// TwinCAT 3 PLC project ScatterSlits
// ProgramVersion: 3.1.4022.3
// libraries:
//   Tc2_MC2, * (Beckhoff Automation GmbH)
//   Tc2_Standard, * (Beckhoff Automation GmbH)
//   Tc2_System, * (Beckhoff Automation GmbH)
//   Tc3_Module, * (Beckhoff Automation GmbH)
// project tree:
//   DUTs/ DUT_M.TcDUT, E_HomeState.TcDUT (not stored), MoveState_t.TcDUT
//   / PlcTask.TcTTO
//   POUs/ FB_Home.TcPOU, FB_HomeToSwitch.TcPOU, FB_Motion.TcPOU, MAIN.TcPOU
// real-time tasks:
//   TASK PlcTask: cycle T#10ms, priority 20, ADS port 350
// motion (NC):
//   TASK NC-Task 1 SAF: cycle T#2ms, priority 4, ADS port 501
//   TASK NC-Task 1 SVB: cycle T#10ms, priority 8, ADS port 511
//   AXIS Axis 1 (id 1)
//     Velo: Maximum=2.2
//     OtherSettings: AllowMotionCmdToSlave=true
//     encoder EncType=4
//       EncPara: MaxCount=#x0000ffff
//         SoftEndMinControl: Range=0.05
//         Inc: RefSoftSyncMask=#x0000ffff
//     drive DrvType=24
//       Analog: VeloReferenz=2, ScaleFactorActTorque=0.1
//       TimeComp: TaskDelayCycles=1
//     controller CtrType=1
//       CtrPara: PriorControlFactor=1
//         PosDiffControl: Range=0.05
//         Observer: BandWidth=20
//   AXIS Axis 2 (id 2)
//     Velo: Maximum=2.2
//     OtherSettings: AllowMotionCmdToSlave=true
//     encoder EncType=4
//       EncPara: Inverse=true, MaxCount=#x0000ffff
//         Inc: RefSoftSyncMask=#x0000ffff
//     drive DrvType=24
//       Analog: VeloReferenz=2, ScaleFactorActTorque=0.1
//       TimeComp: TaskDelayCycles=1
//     controller CtrType=1
//       CtrPara: PriorControlFactor=1
//         PosDiffControl: Range=0.05
//         Observer: BandWidth=20
//   AXIS Axis 3 (id 3)
//     Velo: Maximum=2.2
//     OtherSettings: AllowMotionCmdToSlave=true
//     encoder EncType=4
//       EncPara: Inverse=true, MaxCount=#x0000ffff
//         Inc: RefSoftSyncMask=#x0000ffff
//     drive DrvType=24
//       Analog: VeloReferenz=2, ScaleFactorActTorque=0.1
//       TimeComp: TaskDelayCycles=1
//     controller CtrType=1
//       CtrPara: PriorControlFactor=1
//         PosDiffControl: Range=0.1
//         Observer: BandWidth=20
//   AXIS Axis 4 (id 4)
//     Velo: Maximum=2.2
//     OtherSettings: AllowMotionCmdToSlave=true
//     encoder EncType=4
//       EncPara: MaxCount=#x0000ffff
//         Inc: RefSoftSyncMask=#x0000ffff
//     drive DrvType=24
//       Analog: VeloReferenz=2, ScaleFactorActTorque=0.1
//       TimeComp: TaskDelayCycles=1
//     controller CtrType=1
//       CtrPara: PriorControlFactor=1
//         PosDiffControl: Range=0.1
//         Observer: BandWidth=20
// I/O:
//   DEVICE Device 1 (EtherCAT), AmsNetId 134.79.81.23.2.1
//     Term 1 (EK1100) [EK1100 EtherCAT Coupler (2A E-Bus)]
//       M1  (EL7031) [EL7031 1Ch. Stepper motor output stage (24V, 1.5A)]
//       E1(EL5101) [EL5101 1Ch. Inc. Encoder 5V]
//       M2 (EL7031) [EL7031 1Ch. Stepper motor output stage (24V, 1.5A)]
//       E2 (EL5101) [EL5101 1Ch. Inc. Encoder 5V]
//       M3 (EL7031) [EL7031 1Ch. Stepper motor output stage (24V, 1.5A)]
//       E3 (EL5101) [EL5101 1Ch. Inc. Encoder 5V]
//       M4 (EL7031) [EL7031 1Ch. Stepper motor output stage (24V, 1.5A)]
//       E4 (EL5101) [EL5101 1Ch. Inc. Encoder 5V]
//       Term 10 (EL9011) [EL9011 End Terminal]
// variable links:
//   NC-Task 1 SAF/Axes/Axis 1 <-> Device 1 (EtherCAT)/Term 1 (EK1100)/E1(EL5101)
//     Enc/Inputs/In/nDataIn1[0] <-> ENC Status compact/Counter value
//     Enc/Inputs/In/nDataIn2[0] <-> ENC Status compact/Latch value
//     Enc/Inputs/In/nState1 @bit 4 <-> ENC Status compact/Status/Counter overflow
//     Enc/Inputs/In/nState1 @bit 3 <-> ENC Status compact/Status/Counter underflow
//     Enc/Inputs/In/nState1 @bit 7 <-> ENC Status compact/Status/Extrapolation stall
//     Enc/Inputs/In/nState1 <-> ENC Status compact/Status/Latch C valid
//     Enc/Inputs/In/nState1 @bit 1 <-> ENC Status compact/Status/Latch extern valid
//     Enc/Inputs/In/nState1 @bit 6 <-> ENC Status compact/Status/Open circuit
//     Enc/Inputs/In/nState1 @bit 2 <-> ENC Status compact/Status/Set counter done
//     Enc/Inputs/In/nState1 @bit 5 <-> ENC Status compact/Status/Status of input status
//     Enc/Inputs/In/nState2 @bit 4 <-> ENC Status compact/Status/Status of extern latch
//     Enc/Inputs/In/nState2 <-> ENC Status compact/Status/Status of input A
//     Enc/Inputs/In/nState2 @bit 1 <-> ENC Status compact/Status/Status of input B
//     Enc/Inputs/In/nState2 @bit 2 <-> ENC Status compact/Status/Status of input C
//     Enc/Inputs/In/nState2 @bit 3 <-> ENC Status compact/Status/Status of input gate
//     Enc/Inputs/In/nState2 @bit 5 <-> ENC Status compact/Status/Sync error
//     Enc/Inputs/In/nState2 @bit 6 <-> ENC Status compact/Status/TxPDO State
//     Enc/Inputs/In/nState2 @bit 7 <-> ENC Status compact/Status/TxPDO Toggle
//     Enc/Inputs/In/nState4 @bit 1 <-> WcState/InputToggle
//     Enc/Inputs/In/nState4 <-> WcState/WcState
//     Enc/Outputs/Out/nCtrl1 <-> ENC Control compact/Control/Enable latch C
//     Enc/Outputs/Out/nCtrl1 @bit 3 <-> ENC Control compact/Control/Enable latch extern on negative edge
//     Enc/Outputs/Out/nCtrl1 @bit 1 <-> ENC Control compact/Control/Enable latch extern on positive edge
//     Enc/Outputs/Out/nCtrl1 @bit 2 <-> ENC Control compact/Control/Set counter
//     Enc/Outputs/Out/nDataOut1[0] <-> ENC Control compact/Set counter value
//   NC-Task 1 SAF/Axes/Axis 1 <-> Device 1 (EtherCAT)/Term 1 (EK1100)/M1  (EL7031)
//     Drive/Inputs/In/nState1 @bit 3 <-> STM Status/Status/Error
//     Drive/Inputs/In/nState1 @bit 5 <-> STM Status/Status/Moving negative
//     Drive/Inputs/In/nState1 @bit 4 <-> STM Status/Status/Moving positive
//     Drive/Inputs/In/nState1 @bit 1 <-> STM Status/Status/Ready
//     Drive/Inputs/In/nState1 <-> STM Status/Status/Ready to enable
//     Drive/Inputs/In/nState1 @bit 6 <-> STM Status/Status/Torque reduced
//     Drive/Inputs/In/nState1 @bit 2 <-> STM Status/Status/Warning
//     Drive/Inputs/In/nState2 @bit 5 <-> STM Status/Status/Sync error
//     Drive/Inputs/In/nState2 @bit 7 <-> STM Status/Status/TxPDO Toggle
//     Drive/Inputs/In/nState4 @bit 1 <-> WcState/InputToggle
//     Drive/Inputs/In/nState4 <-> WcState/WcState
//     Drive/Outputs/Out/nCtrl1 <-> STM Control/Control/Enable
//     Drive/Outputs/Out/nCtrl1 @bit 2 <-> STM Control/Control/Reduce torque
//     Drive/Outputs/Out/nCtrl1 @bit 1 <-> STM Control/Control/Reset
//     Drive/Outputs/Out/nDataOut2[0] <-> STM Velocity/Velocity
//   NC-Task 1 SAF/Axes/Axis 2 <-> Device 1 (EtherCAT)/Term 1 (EK1100)/E2 (EL5101)
//     Enc/Inputs/In/nDataIn1[0] <-> ENC Status compact/Counter value
//     Enc/Inputs/In/nDataIn2[0] <-> ENC Status compact/Latch value
//     Enc/Inputs/In/nState1 @bit 4 <-> ENC Status compact/Status/Counter overflow
//     Enc/Inputs/In/nState1 @bit 3 <-> ENC Status compact/Status/Counter underflow
//     Enc/Inputs/In/nState1 @bit 7 <-> ENC Status compact/Status/Extrapolation stall
//     Enc/Inputs/In/nState1 <-> ENC Status compact/Status/Latch C valid
//     Enc/Inputs/In/nState1 @bit 1 <-> ENC Status compact/Status/Latch extern valid
//     Enc/Inputs/In/nState1 @bit 6 <-> ENC Status compact/Status/Open circuit
//     Enc/Inputs/In/nState1 @bit 2 <-> ENC Status compact/Status/Set counter done
//     Enc/Inputs/In/nState1 @bit 5 <-> ENC Status compact/Status/Status of input status
//     Enc/Inputs/In/nState2 @bit 4 <-> ENC Status compact/Status/Status of extern latch
//     Enc/Inputs/In/nState2 <-> ENC Status compact/Status/Status of input A
//     Enc/Inputs/In/nState2 @bit 1 <-> ENC Status compact/Status/Status of input B
//     Enc/Inputs/In/nState2 @bit 2 <-> ENC Status compact/Status/Status of input C
//     Enc/Inputs/In/nState2 @bit 3 <-> ENC Status compact/Status/Status of input gate
//     Enc/Inputs/In/nState2 @bit 5 <-> ENC Status compact/Status/Sync error
//     Enc/Inputs/In/nState2 @bit 6 <-> ENC Status compact/Status/TxPDO State
//     Enc/Inputs/In/nState2 @bit 7 <-> ENC Status compact/Status/TxPDO Toggle
//     Enc/Inputs/In/nState4 @bit 1 <-> WcState/InputToggle
//     Enc/Inputs/In/nState4 <-> WcState/WcState
//     Enc/Outputs/Out/nCtrl1 <-> ENC Control compact/Control/Enable latch C
//     Enc/Outputs/Out/nCtrl1 @bit 3 <-> ENC Control compact/Control/Enable latch extern on negative edge
//     Enc/Outputs/Out/nCtrl1 @bit 1 <-> ENC Control compact/Control/Enable latch extern on positive edge
//     Enc/Outputs/Out/nCtrl1 @bit 2 <-> ENC Control compact/Control/Set counter
//     Enc/Outputs/Out/nDataOut1[0] <-> ENC Control compact/Set counter value
//   NC-Task 1 SAF/Axes/Axis 2 <-> Device 1 (EtherCAT)/Term 1 (EK1100)/M2 (EL7031)
//     Drive/Inputs/In/nState1 @bit 3 <-> STM Status/Status/Error
//     Drive/Inputs/In/nState1 @bit 5 <-> STM Status/Status/Moving negative
//     Drive/Inputs/In/nState1 @bit 4 <-> STM Status/Status/Moving positive
//     Drive/Inputs/In/nState1 @bit 1 <-> STM Status/Status/Ready
//     Drive/Inputs/In/nState1 <-> STM Status/Status/Ready to enable
//     Drive/Inputs/In/nState1 @bit 6 <-> STM Status/Status/Torque reduced
//     Drive/Inputs/In/nState1 @bit 2 <-> STM Status/Status/Warning
//     Drive/Inputs/In/nState2 @bit 5 <-> STM Status/Status/Sync error
//     Drive/Inputs/In/nState2 @bit 7 <-> STM Status/Status/TxPDO Toggle
//     Drive/Inputs/In/nState4 @bit 1 <-> WcState/InputToggle
//     Drive/Inputs/In/nState4 <-> WcState/WcState
//     Drive/Outputs/Out/nCtrl1 <-> STM Control/Control/Enable
//     Drive/Outputs/Out/nCtrl1 @bit 2 <-> STM Control/Control/Reduce torque
//     Drive/Outputs/Out/nCtrl1 @bit 1 <-> STM Control/Control/Reset
//     Drive/Outputs/Out/nDataOut2[0] <-> STM Velocity/Velocity
//   NC-Task 1 SAF/Axes/Axis 3 <-> Device 1 (EtherCAT)/Term 1 (EK1100)/E3 (EL5101)
//     Enc/Inputs/In/nDataIn1[0] <-> ENC Status compact/Counter value
//     Enc/Inputs/In/nDataIn2[0] <-> ENC Status compact/Latch value
//     Enc/Inputs/In/nState1 @bit 4 <-> ENC Status compact/Status/Counter overflow
//     Enc/Inputs/In/nState1 @bit 3 <-> ENC Status compact/Status/Counter underflow
//     Enc/Inputs/In/nState1 @bit 7 <-> ENC Status compact/Status/Extrapolation stall
//     Enc/Inputs/In/nState1 <-> ENC Status compact/Status/Latch C valid
//     Enc/Inputs/In/nState1 @bit 1 <-> ENC Status compact/Status/Latch extern valid
//     Enc/Inputs/In/nState1 @bit 6 <-> ENC Status compact/Status/Open circuit
//     Enc/Inputs/In/nState1 @bit 2 <-> ENC Status compact/Status/Set counter done
//     Enc/Inputs/In/nState1 @bit 5 <-> ENC Status compact/Status/Status of input status
//     Enc/Inputs/In/nState2 @bit 4 <-> ENC Status compact/Status/Status of extern latch
//     Enc/Inputs/In/nState2 <-> ENC Status compact/Status/Status of input A
//     Enc/Inputs/In/nState2 @bit 1 <-> ENC Status compact/Status/Status of input B
//     Enc/Inputs/In/nState2 @bit 2 <-> ENC Status compact/Status/Status of input C
//     Enc/Inputs/In/nState2 @bit 3 <-> ENC Status compact/Status/Status of input gate
//     Enc/Inputs/In/nState2 @bit 5 <-> ENC Status compact/Status/Sync error
//     Enc/Inputs/In/nState2 @bit 6 <-> ENC Status compact/Status/TxPDO State
//     Enc/Inputs/In/nState2 @bit 7 <-> ENC Status compact/Status/TxPDO Toggle
//     Enc/Inputs/In/nState4 @bit 1 <-> WcState/InputToggle
//     Enc/Inputs/In/nState4 <-> WcState/WcState
//     Enc/Outputs/Out/nCtrl1 <-> ENC Control compact/Control/Enable latch C
//     Enc/Outputs/Out/nCtrl1 @bit 3 <-> ENC Control compact/Control/Enable latch extern on negative edge
//     Enc/Outputs/Out/nCtrl1 @bit 1 <-> ENC Control compact/Control/Enable latch extern on positive edge
//     Enc/Outputs/Out/nCtrl1 @bit 2 <-> ENC Control compact/Control/Set counter
//     Enc/Outputs/Out/nDataOut1[0] <-> ENC Control compact/Set counter value
//   NC-Task 1 SAF/Axes/Axis 3 <-> Device 1 (EtherCAT)/Term 1 (EK1100)/M3 (EL7031)
//     Drive/Inputs/In/nState1 @bit 3 <-> STM Status/Status/Error
//     Drive/Inputs/In/nState1 @bit 5 <-> STM Status/Status/Moving negative
//     Drive/Inputs/In/nState1 @bit 4 <-> STM Status/Status/Moving positive
//     Drive/Inputs/In/nState1 @bit 1 <-> STM Status/Status/Ready
//     Drive/Inputs/In/nState1 <-> STM Status/Status/Ready to enable
//     Drive/Inputs/In/nState1 @bit 6 <-> STM Status/Status/Torque reduced
//     Drive/Inputs/In/nState1 @bit 2 <-> STM Status/Status/Warning
//     Drive/Inputs/In/nState2 @bit 5 <-> STM Status/Status/Sync error
//     Drive/Inputs/In/nState2 @bit 7 <-> STM Status/Status/TxPDO Toggle
//     Drive/Inputs/In/nState4 @bit 1 <-> WcState/InputToggle
//     Drive/Inputs/In/nState4 <-> WcState/WcState
//     Drive/Outputs/Out/nCtrl1 <-> STM Control/Control/Enable
//     Drive/Outputs/Out/nCtrl1 @bit 2 <-> STM Control/Control/Reduce torque
//     Drive/Outputs/Out/nCtrl1 @bit 1 <-> STM Control/Control/Reset
//     Drive/Outputs/Out/nDataOut2[0] <-> STM Velocity/Velocity
//   NC-Task 1 SAF/Axes/Axis 4 <-> Device 1 (EtherCAT)/Term 1 (EK1100)/E4 (EL5101)
//     Enc/Inputs/In/nDataIn1[0] <-> ENC Status compact/Counter value
//     Enc/Inputs/In/nDataIn2[0] <-> ENC Status compact/Latch value
//     Enc/Inputs/In/nState1 @bit 4 <-> ENC Status compact/Status/Counter overflow
//     Enc/Inputs/In/nState1 @bit 3 <-> ENC Status compact/Status/Counter underflow
//     Enc/Inputs/In/nState1 @bit 7 <-> ENC Status compact/Status/Extrapolation stall
//     Enc/Inputs/In/nState1 <-> ENC Status compact/Status/Latch C valid
//     Enc/Inputs/In/nState1 @bit 1 <-> ENC Status compact/Status/Latch extern valid
//     Enc/Inputs/In/nState1 @bit 6 <-> ENC Status compact/Status/Open circuit
//     Enc/Inputs/In/nState1 @bit 2 <-> ENC Status compact/Status/Set counter done
//     Enc/Inputs/In/nState1 @bit 5 <-> ENC Status compact/Status/Status of input status
//     Enc/Inputs/In/nState2 @bit 4 <-> ENC Status compact/Status/Status of extern latch
//     Enc/Inputs/In/nState2 <-> ENC Status compact/Status/Status of input A
//     Enc/Inputs/In/nState2 @bit 1 <-> ENC Status compact/Status/Status of input B
//     Enc/Inputs/In/nState2 @bit 2 <-> ENC Status compact/Status/Status of input C
//     Enc/Inputs/In/nState2 @bit 3 <-> ENC Status compact/Status/Status of input gate
//     Enc/Inputs/In/nState2 @bit 5 <-> ENC Status compact/Status/Sync error
//     Enc/Inputs/In/nState2 @bit 6 <-> ENC Status compact/Status/TxPDO State
//     Enc/Inputs/In/nState2 @bit 7 <-> ENC Status compact/Status/TxPDO Toggle
//     Enc/Inputs/In/nState4 @bit 1 <-> WcState/InputToggle
//     Enc/Inputs/In/nState4 <-> WcState/WcState
//     Enc/Outputs/Out/nCtrl1 <-> ENC Control compact/Control/Enable latch C
//     Enc/Outputs/Out/nCtrl1 @bit 3 <-> ENC Control compact/Control/Enable latch extern on negative edge
//     Enc/Outputs/Out/nCtrl1 @bit 1 <-> ENC Control compact/Control/Enable latch extern on positive edge
//     Enc/Outputs/Out/nCtrl1 @bit 2 <-> ENC Control compact/Control/Set counter
//     Enc/Outputs/Out/nDataOut1[0] <-> ENC Control compact/Set counter value
//   NC-Task 1 SAF/Axes/Axis 4 <-> Device 1 (EtherCAT)/Term 1 (EK1100)/M4 (EL7031)
//     Drive/Inputs/In/nState1 @bit 3 <-> STM Status/Status/Error
//     Drive/Inputs/In/nState1 @bit 5 <-> STM Status/Status/Moving negative
//     Drive/Inputs/In/nState1 @bit 4 <-> STM Status/Status/Moving positive
//     Drive/Inputs/In/nState1 @bit 1 <-> STM Status/Status/Ready
//     Drive/Inputs/In/nState1 <-> STM Status/Status/Ready to enable
//     Drive/Inputs/In/nState1 @bit 6 <-> STM Status/Status/Torque reduced
//     Drive/Inputs/In/nState1 @bit 2 <-> STM Status/Status/Warning
//     Drive/Inputs/In/nState2 @bit 5 <-> STM Status/Status/Sync error
//     Drive/Inputs/In/nState2 @bit 7 <-> STM Status/Status/TxPDO Toggle
//     Drive/Inputs/In/nState4 @bit 1 <-> WcState/InputToggle
//     Drive/Inputs/In/nState4 <-> WcState/WcState
//     Drive/Outputs/Out/nCtrl1 <-> STM Control/Control/Enable
//     Drive/Outputs/Out/nCtrl1 @bit 2 <-> STM Control/Control/Reduce torque
//     Drive/Outputs/Out/nCtrl1 @bit 1 <-> STM Control/Control/Reset
//     Drive/Outputs/Out/nDataOut2[0] <-> STM Velocity/Velocity
//   ScatterSlits/ScatterSlits Instance <-> Device 1 (EtherCAT)/Term 1 (EK1100)/M1  (EL7031)
//     PlcTask Inputs/MAIN.M1.LimIn <-> STM Status/Status/Digital input 2
//     PlcTask Inputs/MAIN.M1.LimOut <-> STM Status/Status/Digital input 1
//   ScatterSlits/ScatterSlits Instance <-> Device 1 (EtherCAT)/Term 1 (EK1100)/M2 (EL7031)
//     PlcTask Inputs/MAIN.M2.LimIn <-> STM Status/Status/Digital input 2
//     PlcTask Inputs/MAIN.M2.LimOut <-> STM Status/Status/Digital input 1
//   ScatterSlits/ScatterSlits Instance <-> Device 1 (EtherCAT)/Term 1 (EK1100)/M3 (EL7031)
//     PlcTask Inputs/MAIN.M3.LimIn <-> STM Status/Status/Digital input 2
//     PlcTask Inputs/MAIN.M3.LimOut <-> STM Status/Status/Digital input 1
//   ScatterSlits/ScatterSlits Instance <-> Device 1 (EtherCAT)/Term 1 (EK1100)/M4 (EL7031)
//     PlcTask Inputs/MAIN.M4.LimIn <-> STM Status/Status/Digital input 2
//     PlcTask Inputs/MAIN.M4.LimOut <-> STM Status/Status/Digital input 1
//   ScatterSlits/ScatterSlits Instance <-> NC-Task 1 SAF/Axes/Axis 1
//     PlcTask Inputs/MAIN.Axis1.NcToPlc <-> Outputs/ToPlc
//     PlcTask Outputs/MAIN.Axis1.PlcToNc <-> Inputs/FromPlc
//   ScatterSlits/ScatterSlits Instance <-> NC-Task 1 SAF/Axes/Axis 2
//     PlcTask Inputs/MAIN.Axis2.NcToPlc <-> Outputs/ToPlc
//     PlcTask Outputs/MAIN.Axis2.PlcToNc <-> Inputs/FromPlc
//   ScatterSlits/ScatterSlits Instance <-> NC-Task 1 SAF/Axes/Axis 3
//     PlcTask Inputs/MAIN.Axis3.NcToPlc <-> Outputs/ToPlc
//     PlcTask Outputs/MAIN.Axis3.PlcToNc <-> Inputs/FromPlc
//   ScatterSlits/ScatterSlits Instance <-> NC-Task 1 SAF/Axes/Axis 4
//     PlcTask Inputs/MAIN.Axis4.NcToPlc <-> Outputs/ToPlc
//     PlcTask Outputs/MAIN.Axis4.PlcToNc <-> Inputs/FromPlc

CONFIGURATION ScatterSlits
    RESOURCE PLC ON TwinCAT3
        TASK PlcTask(INTERVAL := T#10ms, PRIORITY := 20);
        PROGRAM MAIN WITH PlcTask : MAIN;
    END_RESOURCE
END_CONFIGURATION

// ---- DUTs/DUT_M.TcDUT
TYPE DUT_M :
STRUCT
	LimOut  At %I* : BOOL;
LimIn At %I* : BOOL;
Encoder At %I* : UINT;
Enable: BOOL;
END_STRUCT

END_TYPE

// ---- DUTs/MoveState_t.TcDUT
TYPE MoveState_t :
(
	MOVESTATE_INIT,
	MOVESTATE_ENABLE,
	MOVESTATE_COUPLE,
	MOVESTATE_DECOUPLE,
	MOVESTATE_FORWARD1,
	MOVESTATE_FORWARD2,
	MOVESTATE_BACKWARDS,
	MOVESTATE_COUPLE2,
	MOVESTATE_HALTSLAVE,
	MOVESTATE_ERROR,
	MOVESTATE_RESET
) UDINT;
END_TYPE

// ---- POUs/MAIN.TcPOU
PROGRAM MAIN
VAR
	
i : INT;
couple:bool;
P1: MC_POWER;
Axis1 : AXIS_REF;
P2: MC_POWER;
Axis2 : AXIS_REF;
P3: MC_POWER;
Axis3 : AXIS_REF;
P4: MC_POWER;
Axis4 : AXIS_REF;


M1:DUT_M;
M2:DUT_M;
M3:DUT_M;
M4:DUT_M;

GearIn: MC_GearIn;
GearInOut: ST_McOutputs;
GearOut: MC_GearOut;
GearOutOut: ST_McOutputs;
//X_Axes : FB_Motion();
//Y_Axes : FB_Motion();

x_go: bool;
y_go:bool;
END_VAR

i:=i+1;
//ignore naming lim in and limout
P1(
	Axis:= Axis1 , 
	Enable:= M1.Enable, 
	Enable_Positive:=M1.LimIn, //FFW DI2
	Enable_Negative:= M1.LimOut, 
	Override:= , 
	BufferMode:= , 
	Options:= , 
	Status=> , 
	Busy=> , 
	Active=> , 
	Error=> , 
	ErrorID=> );

P2(
	Axis:= Axis2 , 
	Enable:= M2.Enable, 
	Enable_Positive:=M2.LimIn  , //FFW Di2
	Enable_Negative:= M2.LimOut , 
	Override:= , 
	BufferMode:= , 
	Options:= , 
	Status=> , 
	Busy=> , 
	Active=> , 
	Error=> , 
	ErrorID=> );


P3(
	Axis:= Axis3 , 
	Enable:= M3.Enable, 
	Enable_Positive:= M3.LimOut  ,  //DI1
	Enable_Negative:= M3.LimIn, 
	Override:= , 
	BufferMode:= , 
	Options:= , 
	Status=> , 
	Busy=> , 
	Active=> , 
	Error=> , 
	ErrorID=> );

P4(
	Axis:= Axis4 , 
	Enable:= M4.Enable, 
	Enable_Positive:=M4.LimOut , //DI1
	Enable_Negative:= M4.LimIn, //DI 2 clse to motor fbw cw
	Override:= , 
	BufferMode:= , 
	Options:= , 
	Status=> , 
	Busy=> , 
	Active=> , 
	Error=> , 
	ErrorID=> );
	
Axis1();
Axis2();
Axis3();
Axis4();

(*
if couple then
	GearIn.Execute := TRUE;
	couple:=false;
	IF GearIn.InGear THEN
				GearIn.Execute := FALSE;
			ELSIF GearIn.Error THEN
				//state := MOVESTATE_ERROR;
			END_IF
END_IF
	
//GearOut(
		
ActCouple();
GearIn.RatioNumerator :=1;
GearIn.RatioDenominator :=1;

X_Axes(Master:= Axis3, Slave:=Axis4, PowerMaster:=P3, PowerSlave:=P4, GO:= x_go);
Y_Axes(Master:= Axis1, Slave:=Axis2, PowerMaster:=P1, PowerSlave:=P2, GO:= y_go);*)

ACTION ActCouple:
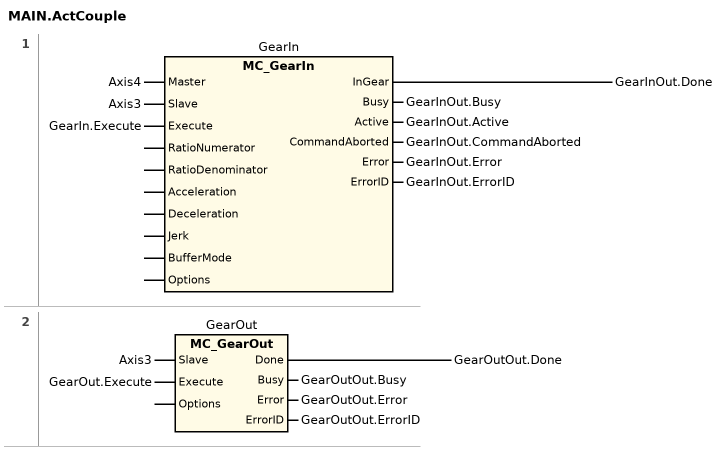
// NETWORK 1
GearIn(
    Master := Axis4,
    Slave := Axis3,
    Execute := GearIn.Execute,
    Busy => GearInOut.Busy,
    Active => GearInOut.Active,
    CommandAborted => GearInOut.CommandAborted,
    Error => GearInOut.Error,
    ErrorID => GearInOut.ErrorID); // MC_GearIn
GearInOut.Done := GearIn.InGear;

// NETWORK 2
GearOut(
    Slave := Axis3,
    Execute := GearOut.Execute,
    Busy => GearOutOut.Busy,
    Error => GearOutOut.Error,
    ErrorID => GearOutOut.ErrorID); // MC_GearOut
GearOutOut.Done := GearOut.Done;
END_ACTION

END_PROGRAM

// ---- POUs/FB_Home.TcPOU
FUNCTION_BLOCK FB_Home
VAR_IN_OUT
	Axis :AXIS_REF;
	fbPowerAxis : MC_POWER;
END_VAR
VAR_INPUT
	bHome: Bool;
END_VAR
VAR
	

	// Homing Functions
	bGo:BOOL := FALSE; //to execute motion
	bIsHomed:BOOL :=FALSE; // should be set to true
	bEnable:Bool; //to be removed
	fbMoveRel: MC_MoveRelative;
	fbSetPosition: MC_SetPosition;
	fbWriteParameter: MC_WriteBoolParameter;
	HomeState: E_HomeState;
	
	fbReset: MC_Reset;
	rHomingDistance : REAL :=-1; 
	rHomingVelocity : REAL :=0.1;
END_VAR



CASE HomeState OF
	H_READY:
		fbSetPosition.Execute := FALSE;
		fbWriteParameter.Execute := FALSE;
		fbMoveRel.Execute := FALSE;
		
		IF (bHome) THEN 
			bHome := FALSE;
			HomeState := H_INIT; 
		END_IF;
	
	H_INIT:
	HomeState:=H_RESET_LL;

		
	H_RESET_LL:
		// disable soft limits in order to be able to move the drive
		fbWriteParameter.ParameterNumber := MC_AxisParameter.EnableLimitNeg;
		fbWriteParameter.Value := FALSE;
		fbWriteParameter.Execute := TRUE;
		if (fbWriteParameter.Done) THEN
			fbWriteParameter.Execute := FALSE;
			HomeState:= H_RESET_HL; 
		END_IF
		
	H_RESET_HL:
		// disable soft limits in order to be able to move the drive
		fbWriteParameter.ParameterNumber := MC_AxisParameter.EnableLimitPos;
		fbWriteParameter.Value := FALSE;
		fbWriteParameter.Execute := TRUE;
		if (fbWriteParameter.Done) THEN
			fbWriteParameter.Execute := FALSE;
			HomeState:= H_ENABLE; 
		END_IF
		
	H_ENABLE:
		// Make Sure drive is enabled
		fbPowerAxis.Enable :=  TRUE;
		fbPowerAxis.Enable_Positive := TRUE;
		fbPowerAxis.Enable_Negative := TRUE;
		IF fbPowerAxis.Status THEN
			HomeState:= H_MOVING;
		ELSIF fbPowerAxis.Error THEN
			HomeState := H_ERROR;
		END_IF

	H_MOVING:
		fbMoveRel.Execute := TRUE;
		IF fbMoveRel.Active  THEN
			(* axis is executing job but is not yet finished *)
			fbMoveRel.Execute := FALSE;
			(* leave this state and buffer a second command *)
			HomeState := H_MOVING2;
		ElSIF fbMoveRel.Done THEN
			fbMoveRel.Execute := FALSE;
			HomeState := H_MOVING;//2?
		ELSIF fbMoveRel.CommandAborted OR fbMoveRel.Error THEN
			fbMoveRel.Execute := FALSE;
			HomeState := H_CHECK;
		END_IF
	
	H_MOVING2:
		IF fbMoveRel.CommandAborted OR fbMoveRel.Error THEN
			HomeState := H_CHECK;
		END_IF	
		IF NOT ( Axis.Status.Moving) OR (fbMoveRel.Done) THEN //(fbMoveAxisABS.Done) AND (fbMoveAxisABS2.Done) THEN
			HomeState := H_MOVING;
			fbMoveRel.Execute := FALSE;	
		END_IF
	
	H_CHECK:
		// Check negative limit switch
		IF NOT (fbPowerAxis.Enable_Negative) THEN
			fbReset.Execute := TRUE;
			HomeState := H_RESET;
		ELSE
			HomeState := H_ERROR;
		END_IF
		//Check position lag monitoring error
		(*if (Axis.Status.ErrorID = 16#00004550)THEN 
			//This^.q_stVGP.pv_xReset_SW := TRUE;
			HomeState := H_RESET;
		ELSE
			HomeState := H_ERROR;
		END_IF*)
	
	H_RESET:
		IF fbReset.Done THEN
			HomeState := H_SET_POS;
		END_IF
	
	H_SET_POS:
	 // Set Current Position
		fbSetPosition.Position := 0;
		fbSetPosition.Execute := TRUE;
		IF ( fbSetPosition.Done ) THEN
			fbSetPosition.Execute := FALSE;
			HomeState:= H_WRITE_LL;
		ELSIF (fbSetPosition.Error) THEN
			HomeState := H_ERROR;
		END_IF

	
	H_WRITE_LL:
	// Re Enable the Soft limits	
		fbWriteParameter.ParameterNumber := MC_AxisParameter.AxisEnMinSoftPosLimit;//AxisEnMaxSoftPosLimit;// .AxisEnMinSoftPosLimit;
		fbWriteParameter.Value := TRUE;
		fbWriteParameter.Execute := TRUE;
		if (fbWriteParameter.Done) THEN
			fbWriteParameter.Execute := FALSE;
			HomeState:= H_WRITE_HL; 
		END_IF
		
	H_WRITE_HL:
	// Re Enable the Soft limits	
		fbWriteParameter.ParameterNumber := MC_AxisParameter.AxisEnMaxSoftPosLimit;
		fbWriteParameter.Value := TRUE;
		fbWriteParameter.Execute := TRUE;
		if (fbWriteParameter.Done) THEN
			fbWriteParameter.Execute := FALSE;
			HomeState:= H_DONE; 
		END_IF
		
	
	H_ERROR:
		//taken care of in the axis motion state machine
	H_DONE:
		//taken care of in the axis motion state machine
		bIsHomed := TRUE;
		HomeState:=H_READY;

END_CASE

// Move backward to fully closed
fbMoveRel(
	Axis:= Axis , 
	Execute:= , 
	Distance:= rHomingDistance , 
	Velocity:= rHomingVelocity, 
	Acceleration:= , 
	Deceleration:= , 
	Jerk:= , 
	BufferMode:= MC_BlendingNext, 
	Options:= , 
	Done=> , 
	Busy=> , 
	Active=> , 
	CommandAborted=> , 
	Error=> , 
	ErrorID=> );
	
// Set Encoder Position
fbSetPosition(
	Axis:= Axis , 
	Execute:= , 
	Position:= 0 , 
	Mode:= FALSE, //Absolute
	Options:= , 
	Done=> , 
	Busy=> , 
	Error=> , 
	ErrorID=> );
	
// Write Parameters
fbWriteParameter(
	Axis:= Axis , 
	Execute:= , 
	ParameterNumber:= , 
	Value:= , 
	Done=> , 
	Busy=> , 
	Error=> , 
	ErrorID=> );

	(*AXIS RESET*)
fbReset(
	Axis:= Axis, 
	Execute:= , 
	Done=> , 
	Busy=> , 
	Error=> , 
	ErrorID=> );
	
If ( fbWriteParameter.Error) OR (fbSetPosition.Error)(* OR (fbMoveRel.Error) *)THEN
	HomeState:= H_ERROR; 
END_IF

END_FUNCTION_BLOCK

// ---- POUs/FB_HomeToSwitch.TcPOU
FUNCTION_BLOCK FB_HomeToSwitch
VAR_INPUT
	En: BOOL;
	bReset: BOOL;
    bExecute: BOOL;	
    bCamSensor:BOOL;	
	nSearchDirTwoardsCam: MC_Direction;
	nSearchDirOffCam: MC_Direction;
	fHomePosition:LREAL;	
	fVelocityToCamNC: LREAL; //Velcoity when searching for cam
	fVelocityFromCamNC: LREAL; // Velocity after found cam (searching for next signal transition)
END_VAR
VAR_IN_OUT
	Axis: AXIS_REF;
END_VAR
VAR_OUTPUT
	EnO: BOOL;	
	bBusy: BOOL;
	bDone: BOOL;
	bHomed:BOOL;
	bError: BOOL;
	nErrorId: UDINT;
END_VAR
VAR
	fbHome: MC_Home;	
	fbWriteHomeDirCamToNC:FB_WriteParameterInNc_v1_00;
	fbWriteHomeDirSyncToNC:FB_WriteParameterInNc_v1_00;
	fbWriteHomeModeToNC:FB_WriteParameterInNc_v1_00;
	fbWriteHomeVelocitiesToNC: FB_HomeWriteNcVelocities;
	bConfigNCDone:BOOL:=FALSE;
	fbRTrigg: R_TRIG;
END_VAR

En:=EnO;
IF bReset THEN
	bConfigNCDone:=FALSE;
	bError:=FALSE;
	nErrorId:=0;
END_IF 
	
//Start preparation of NC if rising edge on bExecute
fbRTrigg(CLK:=bExecute);
IF fbRTrigg.Q THEN
	bConfigNCDone:=FALSE;
END_IF

 
fbWriteHomeDirCamToNC(
	bExecute:=bExecute AND NOT bConfigNCDone,
	nDeviceGroup:=16#5000,
	nIndexOffset:=16#101,	//Direction for Calibration Cam Search	
	nData:=BOOL_TO_DWORD(nSearchDirTwoardsCam=MC_Negative_Direction),//BOOL_TO_DWORD(NOT bSearchDirTwoardsCam),
	Axis:=Axis
);

fbWriteHomeDirSyncToNC(
	bExecute:= bExecute AND NOT bConfigNCDone,
	nDeviceGroup:=16#5000 ,
	nIndexOffset:=16#102 , //Direction for Sync Impuls Search
	nData:=BOOL_TO_DWORD(nSearchDirOffCam=MC_Negative_Direction),//BOOL_TO_DWORD(NOT bSearchDirOffCam),
	Axis:= Axis 
);

fbWriteHomeModeToNC(
	bExecute:=bExecute AND NOT bConfigNCDone,
	nDeviceGroup:=16#5000,
	nIndexOffset:=16#107,  //Reference Mode
	nData:=1,
	Axis:=axis);
	
fbWriteHomeVelocitiesToNC(
  En:=En,
  bExecute:=bExecute AND NOT bConfigNCDone,
  bReset:=bReset,
  fVelocityFromCam:=fVelocityFromCamNC,
  fVelocityToCam:=fVelocityToCamNC,
  Axis:=Axis);

fbHome.bCalibrationCam:=bCamSensor;

fbHome(
	Execute:=bExecute AND bConfigNCDone(* AND NOT bError*),
	Position:=fHomePosition,
	HomingMode:=0,
	Axis:=Axis
	);
bBusy:=(fbHome.Busy OR (NOT bConfigNCDone AND bExecute));
bDone:=fbHome.Done AND bConfigNCDone;
bHomed:=Axis.Status.Homed;

IF (NOT bConfigNCDone) AND fbWriteHomeDirCamToNC.bDone AND fbWriteHomeDirSyncToNC.bDone AND fbWriteHomeModeToNC.bDone AND fbWriteHomeVelocitiesToNC.bDone THEN
  bConfigNCDone:=TRUE;
END_IF

//For some reason MC_HOME gives an Error for one cycle of NC-Task 1 SVB (10ms default..) so filter with bExecute
bError:=(fbHome.Error AND bExecute) OR fbWriteHomeDirCamToNC.bError OR fbWriteHomeDirSyncToNC.bError OR fbWriteHomeModeToNC.bError OR fbWriteHomeVelocitiesToNC.bError;

IF (fbHome.Error AND bExecute) THEN
  nErrorId:=fbHome.ErrorID;
ELSIF fbWriteHomeDirCamToNC.bError THEN
  nErrorId:=fbWriteHomeDirCamToNC.nErrorId;
ELSIF fbWriteHomeDirSyncToNC.bError THEN
  nErrorId:=fbWriteHomeDirSyncToNC.nErrorId;
ELSIF fbWriteHomeModeToNC.bError THEN
  nErrorId:=fbWriteHomeModeToNC.nErrorId;
ELSIF fbWriteHomeVelocitiesToNC.bError THEN
  nErrorId:=fbWriteHomeVelocitiesToNC.nErrorId;  
END_IF

END_FUNCTION_BLOCK

// ---- POUs/FB_Motion.TcPOU
FUNCTION_BLOCK FB_Motion
VAR_IN_OUT

/// axis reference data structure 
	Master: AXIS_REF;
	/// axis reference data structure 
	Slave: AXIS_REF;
	PowerMaster: MC_Power;
	PowerSlave: MC_Power;
	GO : BOOL;// := FALSE;
END_VAR
VAR_OUTPUT
END_VAR
VAR

	/// state machine state 
	state: MoveState_t;
	
	/// debug function block output data 
	PowerMasterOut: ST_McOutputs;
	
	/// debug function block output data 
	PowerSlaveOut: ST_McOutputs;
	//MoveMaster: MC_MoveAbsolute;
	/// debug function block output data 
	MoveMasterOut: ST_McOutputs;
	//MoveSlave: MC_MoveAbsolute;
	/// debug function block output data 
	MoveSlaveOut: ST_McOutputs;
	ResetMaster: MC_Reset;
	/// debug function block output data 
	ResetMasterOut: ST_McOutputs;
	ResetSlave: MC_Reset;
	/// debug function block output data 
	ResetSlaveOut: ST_McOutputs;
	GearIn: MC_GearIn;
	GearInOut: ST_McOutputs;
	GearOut: MC_GearOut;
	GearOutOut: ST_McOutputs;
	HaltSlave: MC_Halt;
	HaltSlaveOut: ST_McOutputs;
	
	MoveMaster: MC_MoveRelative;
	MoveSlave: MC_MoveRelative;
END_VAR

	(* update the axis status at the beginning of each cycle *)
	//Master();
	//Slave();
if  NOT (GO) then
	state := MOVESTATE_INIT;	
END_IF
	(* move axis using a state machine *)
	CASE state OF

		MOVESTATE_INIT :	(* initialisation *)
			(* initialize all function blocks *)
			MoveMaster.Execute := FALSE;
			MoveSlave.Execute := FALSE;
			HaltSlave.Execute := FALSE;
			ResetMaster.Execute := FALSE;
			ResetSlave.Execute := FALSE;
			GearIn.Execute := FALSE;
			GearOut.Execute := FALSE;
			if (GO) then
				state := MOVESTATE_ENABLE;	
			END_IF
			

		MOVESTATE_ENABLE :
		//	PowerMaster.Enable := TRUE;
		//	PowerMaster.Enable_Positive := TRUE;
		//	PowerMaster.Enable_Negative := TRUE;
		//	PowerSlave.Enable := TRUE;
		//	PowerSlave.Enable_Positive := TRUE;
		//	PowerSlave.Enable_Negative := TRUE;
			IF PowerMaster.Status AND PowerSlave.Status THEN
				state := MOVESTATE_COUPLE;
			ELSIF PowerMaster.Error OR PowerSlave.Error THEN
				state := MOVESTATE_ERROR;
			END_IF

		MOVESTATE_COUPLE :
			GearIn.Execute := TRUE;
			IF GearIn.InGear THEN
				GearIn.Execute := FALSE;
				state := MOVESTATE_FORWARD1;
			ELSIF GearIn.Error THEN
				state := MOVESTATE_ERROR;
			END_IF

		MOVESTATE_FORWARD1:		(* start to first position *)
			MoveMaster.Distance := 7;		(* start to intermediate target position *)
			MoveMaster.Velocity := 0.3;		(* medium velocity level *)
			MoveMaster.BufferMode := MC_Buffered;
			MoveMaster.Execute := TRUE;
			IF Master.NcToPlc.SetPos > 20 THEN
				state := MOVESTATE_HALTSLAVE;
			ELSIF MoveMaster.Done  THEN
				(* axis is executing job but is not yet finished *)
				MoveMaster.Execute := FALSE;
				state := MOVESTATE_BACKWARDS;
			ELSIF MoveMaster.CommandAborted OR MoveMaster.Error THEN
				state := MOVESTATE_ERROR;
			END_IF

		MOVESTATE_HALTSLAVE :
			(* stopping a slave in motion is possible from TwinCAT 2.11if
			    the parameter "allow motion commands to slaves" is enabled.
			    The slave will automatically be decoupled and stoped.
			*)
			HaltSlave.Execute := TRUE;
			IF HaltSlave.Done AND MoveMaster.Done THEN (* wait for master and slave finished *)
				MoveMaster.Execute := FALSE;
				HaltSlave.Execute := FALSE;
				state := MOVESTATE_COUPLE2;
			ELSIF HaltSlave.Error OR HaltSlave.CommandAborted THEN
				state := MOVESTATE_ERROR;
			ELSIF MoveMaster.CommandAborted OR MoveMaster.Error THEN
				state := MOVESTATE_ERROR;
			END_IF

		MOVESTATE_COUPLE2 :
			GearIn.Execute := TRUE;
			IF GearIn.InGear THEN
				GearIn.Execute := FALSE;
				state := MOVESTATE_FORWARD2;
			ELSIF GearIn.Error THEN
				state := MOVESTATE_ERROR;
			END_IF

		MOVESTATE_FORWARD2 :			(* move to next position *)
			MoveMaster.Distance := 5;		(* start to target position *)
			MoveMaster.Velocity := 0.2;		(* medium velocity level *)
			MoveMaster.BufferMode := MC_Buffered;
			MoveMaster.Execute := TRUE;
			IF Master.NcToPlc.SetPos > 25 THEN
				state := MOVESTATE_DECOUPLE;
			ELSIF MoveMaster.Done  THEN
				(* axis is executing job but is not yet finished *)
				MoveMaster.Execute := FALSE;
				state := MOVESTATE_BACKWARDS;
			ELSIF MoveMaster.CommandAborted OR MoveMaster.Error THEN
				state := MOVESTATE_ERROR;
			END_IF

		MOVESTATE_DECOUPLE :
			(* if a slave is decoupled in motion the axis will continue moving at constant velocity *)
			GearOut.Execute := TRUE;
			IF GearOut.Done AND MoveMaster.Done THEN (* wait for master motion finished *)
				GearOut.Execute := FALSE;
				MoveMaster.Execute := FALSE;
				state := MOVESTATE_BACKWARDS;
			ELSIF GearOut.Error THEN
				state := MOVESTATE_ERROR;
			ELSIF MoveMaster.CommandAborted OR MoveMaster.Error THEN
				state := MOVESTATE_ERROR;
			END_IF

		MOVESTATE_BACKWARDS :	(* move back to initial position *)
			MoveMaster.Distance := -12;		(* position close to initial position *)
			MoveMaster.Velocity := 0.3;		(* high velocity *)
			MoveMaster.Execute := TRUE;
			MoveSlave.Distance := -10;		(* position close to initial position *)
			MoveSlave.Velocity := 0.3;		(* high velocity *)
			MoveSlave.Execute := TRUE;
			IF MoveMaster.Done AND MoveSlave.Done THEN
				(* axis is executing job but is not yet finished *)
				MoveMaster.Execute := FALSE;
				(* leave this state and buffer a second command *)
				state := MOVESTATE_INIT;
			ELSIF MoveMaster.CommandAborted OR MoveMaster.Error
				OR  MoveSlave.CommandAborted OR MoveSlave.Error
				THEN
				state := MOVESTATE_ERROR;
			END_IF

		MOVESTATE_ERROR :
			IF Master.Status.Error OR Slave.Status.Error THEN
				state := MOVESTATE_RESET;	(* axis error requires reset *)
			ELSE
				state := MOVESTATE_INIT;		(* function block errors don't need a reset *)
			END_IF

		MOVESTATE_RESET :
			ResetMaster.Execute := TRUE;
			ResetSlave.Execute := TRUE;
			IF ResetMaster.Done AND ResetSlave.Done THEN
				state := MOVESTATE_INIT;
			ELSIF ResetMaster.Error OR ResetSlave.Error THEN
				state := MOVESTATE_INIT; (* can't do anything here *)
			END_IF

	END_CASE

	//ActPower();		(* call the power function block *)
	ActMoveRel();		(* call the move function block *)
	ActReset();		(* call the reset function block *)
	ActCouple();		(* call the master slave coupling function block *)

ACTION ActCouple:
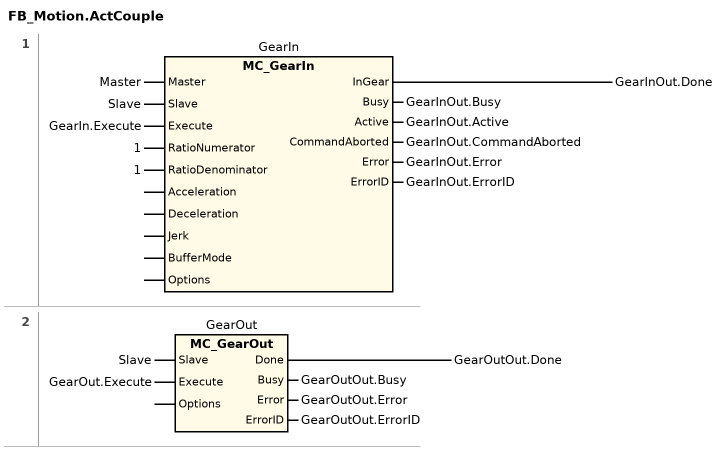
// NETWORK 1
GearIn(
    Master := Master,
    Slave := Slave,
    Execute := GearIn.Execute,
    RatioNumerator := 1,
    RatioDenominator := 1,
    Busy => GearInOut.Busy,
    Active => GearInOut.Active,
    CommandAborted => GearInOut.CommandAborted,
    Error => GearInOut.Error,
    ErrorID => GearInOut.ErrorID); // MC_GearIn
GearInOut.Done := GearIn.InGear;

// NETWORK 2
GearOut(
    Slave := Slave,
    Execute := GearOut.Execute,
    Busy => GearOutOut.Busy,
    Error => GearOutOut.Error,
    ErrorID => GearOutOut.ErrorID); // MC_GearOut
GearOutOut.Done := GearOut.Done;
END_ACTION

ACTION ActMove:
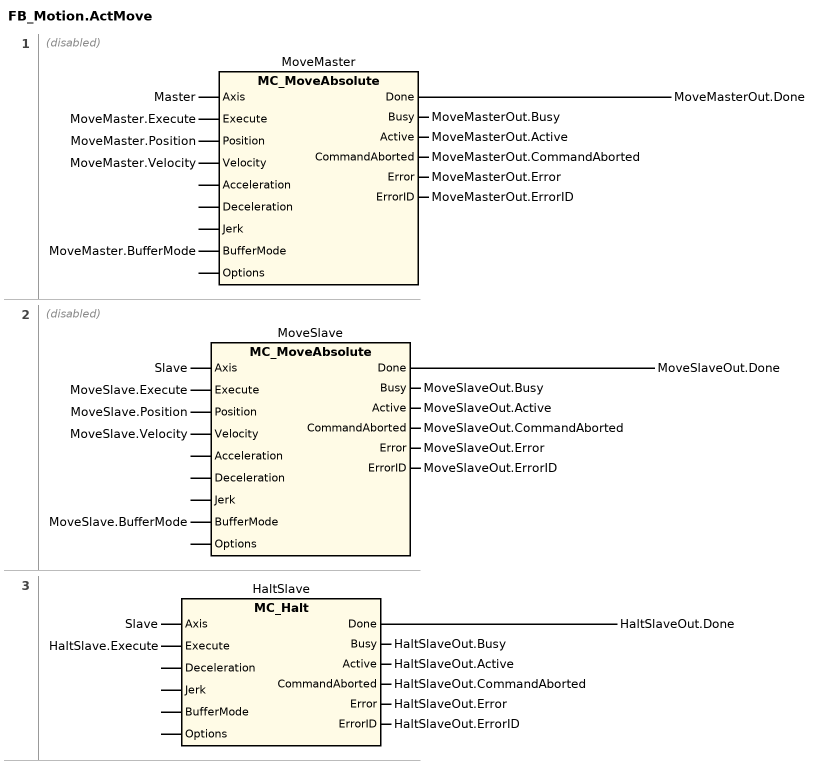
// NETWORK 1 (disabled)
// MoveMaster(
//     Axis := Master,
//     Execute := MoveMaster.Execute,
//     Position := MoveMaster.Position,
//     Velocity := MoveMaster.Velocity,
//     BufferMode := MoveMaster.BufferMode,
//     Busy => MoveMasterOut.Busy,
//     Active => MoveMasterOut.Active,
//     CommandAborted => MoveMasterOut.CommandAborted,
//     Error => MoveMasterOut.Error,
//     ErrorID => MoveMasterOut.ErrorID); // MC_MoveAbsolute
// MoveMasterOut.Done := MoveMaster.Done;

// NETWORK 2 (disabled)
// MoveSlave(
//     Axis := Slave,
//     Execute := MoveSlave.Execute,
//     Position := MoveSlave.Position,
//     Velocity := MoveSlave.Velocity,
//     BufferMode := MoveSlave.BufferMode,
//     Busy => MoveSlaveOut.Busy,
//     Active => MoveSlaveOut.Active,
//     CommandAborted => MoveSlaveOut.CommandAborted,
//     Error => MoveSlaveOut.Error,
//     ErrorID => MoveSlaveOut.ErrorID); // MC_MoveAbsolute
// MoveSlaveOut.Done := MoveSlave.Done;

// NETWORK 3
HaltSlave(
    Axis := Slave,
    Execute := HaltSlave.Execute,
    Busy => HaltSlaveOut.Busy,
    Active => HaltSlaveOut.Active,
    CommandAborted => HaltSlaveOut.CommandAborted,
    Error => HaltSlaveOut.Error,
    ErrorID => HaltSlaveOut.ErrorID); // MC_Halt
HaltSlaveOut.Done := HaltSlave.Done;
END_ACTION

ACTION ActMoveRel:
MoveMaster(
	Axis:= Master , 
	Execute:= , 
	Distance:= , 
	Velocity:= , 
	Acceleration:= , 
	Deceleration:= , 
	Jerk:= , 
	BufferMode:= , 
	Options:= , 
	Done=> MoveMasterOut.Done, 
	Busy=> MoveMasterOut.Busy, 
	Active=> MoveMasterOut.Active , 
	CommandAborted=> MoveMasterOut.CommandAborted , 
	Error=> MoveMasterOut.Error, 
	ErrorID=> MoveMasterOut.ErrorID );
	
MoveSlave(
	Axis:= Slave, 
	Execute:= , 
	Distance:= , 
	Velocity:= , 
	Acceleration:= , 
	Deceleration:= , 
	Jerk:= , 
	BufferMode:= , 
	Options:= , 
	Done=> MoveSlaveOut.Done, 
	Busy=> MoveSlaveOut.Busy, 
	Active=> MoveSlaveOut.Active , 
	CommandAborted=> MoveSlaveOut.CommandAborted , 
	Error=> MoveSlaveOut.Error, 
	ErrorID=> MoveSlaveOut.ErrorID );
END_ACTION

ACTION ActPower:
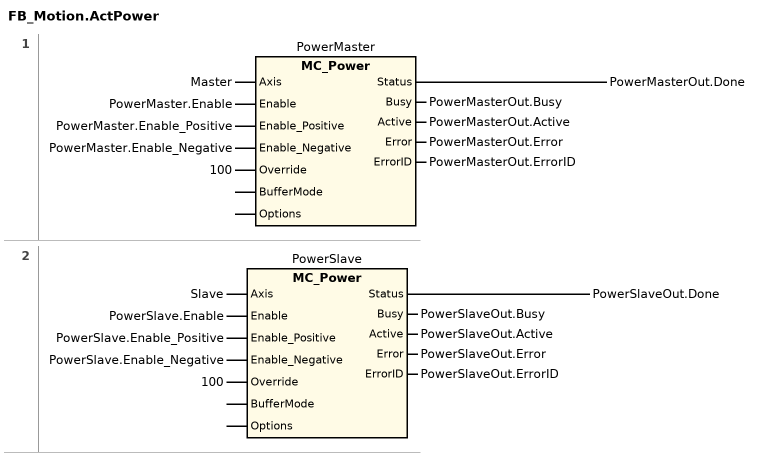
// NETWORK 1
PowerMaster(
    Axis := Master,
    Enable := PowerMaster.Enable,
    Enable_Positive := PowerMaster.Enable_Positive,
    Enable_Negative := PowerMaster.Enable_Negative,
    Override := 100,
    Busy => PowerMasterOut.Busy,
    Active => PowerMasterOut.Active,
    Error => PowerMasterOut.Error,
    ErrorID => PowerMasterOut.ErrorID); // MC_Power
PowerMasterOut.Done := PowerMaster.Status;

// NETWORK 2
PowerSlave(
    Axis := Slave,
    Enable := PowerSlave.Enable,
    Enable_Positive := PowerSlave.Enable_Positive,
    Enable_Negative := PowerSlave.Enable_Negative,
    Override := 100,
    Busy => PowerSlaveOut.Busy,
    Active => PowerSlaveOut.Active,
    Error => PowerSlaveOut.Error,
    ErrorID => PowerSlaveOut.ErrorID); // MC_Power
PowerSlaveOut.Done := PowerSlave.Status;
END_ACTION

ACTION ActReset:
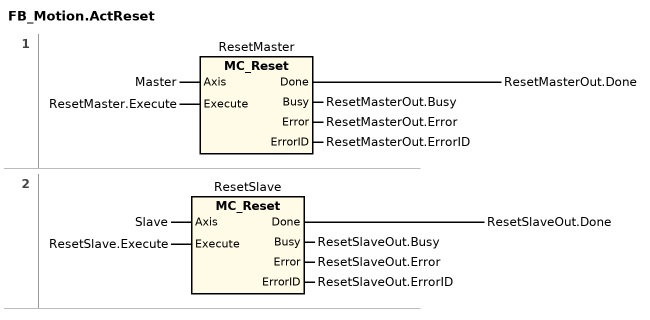
// NETWORK 1
ResetMaster(
    Axis := Master,
    Execute := ResetMaster.Execute,
    Busy => ResetMasterOut.Busy,
    Error => ResetMasterOut.Error,
    ErrorID => ResetMasterOut.ErrorID); // MC_Reset
ResetMasterOut.Done := ResetMaster.Done;

// NETWORK 2
ResetSlave(
    Axis := Slave,
    Execute := ResetSlave.Execute,
    Busy => ResetSlaveOut.Busy,
    Error => ResetSlaveOut.Error,
    ErrorID => ResetSlaveOut.ErrorID); // MC_Reset
ResetSlaveOut.Done := ResetSlave.Done;
END_ACTION

END_FUNCTION_BLOCK
